TYPE ST_GC_ALID :
STRUCT
END_STRUCT
END_TYPE

(* stored: Version 1.1.0.1, ProductVersion 3.1.4026.18
   DUT ST_GC_ALID: Id {9dfbdf1b-d1b9-4d38-80ac-3a0c9425e816} *)
